// Interface consumed by device FBs to interact with the Sparkplug session.
// Decouples device FBs from the concrete FB_SparkplugSession type,
// enabling testability without a live MQTT connection.
INTERFACE I_SparkplugSession

// Returns the current seq counter and advances it (0–255 wrapping).
// Call once per outbound message to stamp the payload header.
METHOD GetNextSeq : ULINT
END_METHOD

// Returns TRUE when the session is in the Online state.
METHOD IsOnline : BOOL
END_METHOD

// Publishes a pre-encoded payload to the broker.
// Only succeeds when the session is Online or Birthing.
METHOD Publish : BOOL
VAR_INPUT
	sTopic		: STRING(255);
	pPayload	: POINTER TO BYTE;
	nLen		: UDINT;
	nQos		: UDINT;
	bRetain		: BOOL;
END_VAR
END_METHOD

// Sparkplug group ID — used by device FBs to build their own topics.
PROPERTY GroupId : STRING(127)
GET
END_GET
END_PROPERTY

// Sparkplug node ID — used by device FBs to build their own topics.
PROPERTY NodeId : STRING(127)
GET
END_GET
END_PROPERTY

END_INTERFACE

(* stored: Version 1.1.0.1
   Itf I_SparkplugSession: Id {22222222-0000-0000-0000-000000000001}, SpecialFunc None
   Method GetNextSeq: Id {22222222-0000-0000-0000-000000000010}
   Method IsOnline: Id {22222222-0000-0000-0000-000000000011}
   Method Publish: Id {22222222-0000-0000-0000-000000000012}
   Property GroupId: Id {22222222-0000-0000-0000-000000000020}
   Get Get: Id {22222222-0000-0000-0000-000000000021}
   Property NodeId: Id {22222222-0000-0000-0000-000000000022}
   Get Get: Id {22222222-0000-0000-0000-000000000023} *)
